SUBAPPLICATION Uebung_008 (* Subapplication Type *)
  (* Standard: 61499-2 *)
  (* Version 1.0, 2023-10-23, franz *)
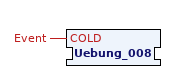
  EVENT_INPUT
    COLD;
  END_EVENT
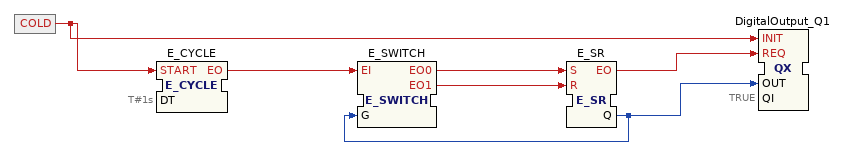
  FBS
    DigitalOutput_Q1 : QX(QI := TRUE);
    E_CYCLE : E_CYCLE(DT := T#1s);
    E_SWITCH : E_SWITCH;
    E_SR : E_SR;
  END_FBS
  EVENT_CONNECTIONS
    COLD TO DigitalOutput_Q1.INIT;
    COLD TO E_CYCLE.START;
    E_CYCLE.EO TO E_SWITCH.EI;
    E_SWITCH.EO0 TO E_SR.S;
    E_SWITCH.EO1 TO E_SR.R;
    E_SR.EO TO DigitalOutput_Q1.REQ;
  END_CONNECTIONS
  DATA_CONNECTIONS
    E_SR.Q TO E_SWITCH.G;
    E_SR.Q TO DigitalOutput_Q1.OUT;
  END_CONNECTIONS
END_SUBAPPLICATION
